// TwinCAT 3 PLC project Untitled1
// ProgramVersion: 3.1.4020.4
// libraries:
//   Tc2_Standard, * (Beckhoff Automation GmbH)
//   Tc2_System, * (Beckhoff Automation GmbH)
//   Tc3_Interfaces, * (Beckhoff Automation GmbH)
//   Tc3_Module, * (Beckhoff Automation GmbH)
// project tree:
//   / PlcTask.TcTTO
//   POUs/ MAIN.TcPOU
// real-time tasks:
//   TASK PlcTask: cycle T#10ms, priority 20, ADS port 350
//   TASK Task 4: cycle T#10ms, priority 1, ADS port 301
// I/O:
//   DEVICE Device 1 (EtherCAT), AmsNetId 192.168.0.231.2.1
//     Term 1 (EK1200) [EK1200-5000 EtherCAT Power supply (2A E-Bus)]
//       Term 2 (EL6900) [EL6900, TwinSAFE PLC]
//       Term 3 (EL1904) [EL1904, 4 Ch. Safety Input 24V, TwinSAFE]
//         modules: Module 1 (FSOES)
//       Term 4 (EL6910) [EL6910, TwinSAFE PLC]
//       Term 5 (EL6930) [EL6930, TwinSAFE PLC]
//       Term 6 [EL9011 End Terminal]
// variable links:
//   Task 4 <-> Device 1 (EtherCAT)/Term 1 (EK1200)/Term 3 (EL1904)
//     Inputs/Var 69 <-> Module 1 (FSOES)/TxPDO/FSOE/FSoE Slave CMD

CONFIGURATION Untitled1
    RESOURCE PLC ON TwinCAT3
        TASK PlcTask(INTERVAL := T#10ms, PRIORITY := 20);
        PROGRAM MAIN WITH PlcTask : MAIN;
    END_RESOURCE
END_CONFIGURATION

// ---- POUs/MAIN.TcPOU
PROGRAM MAIN
VAR
	byByte		AT %MB0 : ARRAY [0..1027] OF BYTE;
	i			: INT;
	moreBytes	: ARRAY [0..8192] OF BYTE;
END_VAR

FOR i := 4 TO 1027 BY 1 DO
	byByte[i] := byByte[i] + 1;
END_FOR

END_PROGRAM
